PROGRAM MAIN
VAR
	fileOpen : FB_FileOpen;
	fileWrite : FB_FileWrite;
	fileClose : FB_FileClose;
	step : DINT := 0;
	handle : UINT;
	buffer : ARRAY[1..10] OF BYTE := [65, 66, 67, 13, 10];
	busy : BOOL;
	error : BOOL;
END_VAR

// write to a file as a simple test
CASE step OF
	0:
		fileOpen(
			sNetId:= '', 
			sPathName:= 'C:\TwinCAT\test.txt', 
			nMode:= FOPEN_MODEWRITE, 
			ePath:= PATH_GENERIC, 
			bExecute:= TRUE, 
			tTimeout:= T#5S, 
			bBusy=> busy, 
			bError=> error, 
			nErrId=> , 
			hFile=> handle);
			
			IF NOT fileOpen.bBusy THEN
				step := step + 1;
			END_IF
			
	1:
			fileOpen(bExecute := FALSE);
			step := step + 1;
	2:
		fileWrite(
			sNetId:= '', 
			hFile:= handle, 
			pWriteBuff:= ADR(buffer), 
			cbWriteLen:= 6, 
			bExecute:= TRUE, 
			tTimeout:= T#5S, 
			bBusy=> busy, 
			bError=> error, 
			nErrId=> , 
			cbWrite=> );
		IF NOT fileWrite.bBusy THEN
			step := step + 1;
		END_IF
	3:
		fileWrite(bExecute := FALSE);
		step := step + 1;
	4:
		fileClose(
			sNetId:= '', 
			hFile:= handle, 
			bExecute:= TRUE, 
			tTimeout:= T#5S, 
			bBusy=> busy, 
			bError=> error, 
			nErrId=> );
		IF NOT fileClose.bBusy THEN
			step := step + 1;
		END_IF
	5:
		fileClose(bExecute := FALSE);
		step := step + 1;
END_CASE

END_PROGRAM

(* stored: Version 1.1.0.1, ProductVersion 3.1.4024.3
   POU MAIN: Id {869cc47a-f229-4c2a-a727-d4b382bc7f7f}, SpecialFunc None *)
